// TwinCAT 3 PLC project SPS
// ProgramVersion: 3.1.4024.0
// libraries:
//   Tc2_MC2, * (Beckhoff Automation GmbH)
//   Tc2_Standard, * (Beckhoff Automation GmbH)
//   Tc2_System, * (Beckhoff Automation GmbH)
//   Tc3_IotBase, * (Beckhoff Automation GmbH)
//   Tc3_Module, * (Beckhoff Automation GmbH)
//   VisuDialogs, * (System)
//   VisuSymbols,3.5.10.0,System
// project tree:
//   DUTs/ eBetriebszustand.TcDUT (not stored)
//   / GlobalTextList.TcGTLO, PlcTask.TcTTO, Visualization Manager.TcVMO (not stored)
//   GVLs/ GVL_PosKinematic.TcGVL (not stored), IFC_HW.TcGVL (not stored)
//   POUs/Abfüllmodul/ FB_Abfuellmodul.TcPOU, FB_Dispenser.TcPOU, FB_EZylinder.TcPOU (not stored), FB_Vereinzelung.TcPOU
//   POUs/Abfüllmodul/Transport/ FB_Foerderband.TcPOU, FB_Transport.TcPOU, FB_Transport_A.TcPOU (not stored), FB_Transport_E.TcPOU (not stored), FB_Transport_Logik.TcPOU
//   POUs/ FUN_Scale.TcPOU (not stored), MAIN.TcPOU
//   POUs/IoT/ FB_MQTT.TcPOU (not stored)
//   POUs/Manipulator/ FB_Manipulator.TcPOU
//   POUs/Manipulator/Roboter/ FB_Roboter.TcPOU, FB_Roboter_Axis.TcPOU, FB_Roboter_E.TcPOU, FB_Roboter_Logik.TcPOU
//   POUs/Statusleuchte/ FB_Ampelleuchte.TcPOU (not stored), FB_Blinklicht.TcPOU (not stored)
//   VISUs/ Visualization.TcVIS
// real-time tasks:
//   TASK PlcTask: cycle T#10ms, priority 20, ADS port 350
// motion (NC):
//   TASK NC-Task 1 SAF: cycle T#2ms, priority 4, ADS port 501
//   TASK NC-Task 1 SVB: cycle T#10ms, priority 8, ADS port 511
//   AXIS Achse_Band (id 1)
//     OtherSettings: AllowMotionCmdToSlave=true
//     encoder EncType=1
//     drive DrvType=5
//       Analog: TorqueSetpointScale=10, ScaleFactorActTorque=0.1
//       TimeComp: TaskDelayCycles=1
//     controller CtrType=1
//       CtrPara: PriorControlFactor=1
//         Observer: BandWidth=20
//   AXIS Achse_Dispenser_Rot (id 2)
//     OtherSettings: AllowMotionCmdToSlave=true
//     encoder EncType=1
//     drive DrvType=5
//       Analog: TorqueSetpointScale=10, ScaleFactorActTorque=0.1
//       TimeComp: TaskDelayCycles=1
//     controller CtrType=1
//       CtrPara: PriorControlFactor=1
//         Observer: BandWidth=20
//   AXIS Achse_Dispenser_Gruen (id 3)
//     OtherSettings: AllowMotionCmdToSlave=true
//     encoder EncType=1
//     drive DrvType=5
//       Analog: TorqueSetpointScale=10, ScaleFactorActTorque=0.1
//       TimeComp: TaskDelayCycles=1
//     controller CtrType=1
//       CtrPara: PriorControlFactor=1
//         Observer: BandWidth=20
//   AXIS Achse_Dispenser_Blau (id 4)
//     OtherSettings: AllowMotionCmdToSlave=true
//     encoder EncType=1
//     drive DrvType=5
//       Analog: TorqueSetpointScale=10, ScaleFactorActTorque=0.1
//       TimeComp: TaskDelayCycles=1
//     controller CtrType=1
//       CtrPara: PriorControlFactor=1
//         Observer: BandWidth=20
//   AXIS Achse_Manipulator_X (id 5)
//     Velo: RefSearch=15, RefSync=15
//     OtherSettings: AllowMotionCmdToSlave=true
//     encoder EncType=1
//       EncPara: ScaleFactorNumerator=0.0025
//         Inc: RefSearchInverse=true, RefSyncInverse=false
//     drive DrvType=5
//       Analog: TorqueSetpointScale=10, ScaleFactorActTorque=0.1
//       TimeComp: TaskDelayCycles=1
//     controller CtrType=1
//       CtrPara: PriorControlFactor=1
//         Observer: BandWidth=20
//   AXIS Achse_Manipulator_Y (id 6)
//     Velo: RefSearch=15, RefSync=15
//     OtherSettings: AllowMotionCmdToSlave=true
//     encoder EncType=1
//       Inc: RefSearchInverse=true, RefSyncInverse=false
//     drive DrvType=5
//       Analog: TorqueSetpointScale=10, ScaleFactorActTorque=0.1
//       TimeComp: TaskDelayCycles=1
//     controller CtrType=1
//       CtrPara: PriorControlFactor=1
//         Observer: BandWidth=20
//   AXIS Achse_Manipulator_Z (id 7)
//     Velo: RefSearch=15, RefSync=15
//     OtherSettings: AllowMotionCmdToSlave=true
//     encoder EncType=1
//       Inc: RefSearchInverse=true, RefSyncInverse=false
//     drive DrvType=5
//       Analog: TorqueSetpointScale=10, ScaleFactorActTorque=0.1
//       TimeComp: TaskDelayCycles=1
//     controller CtrType=1
//       CtrPara: PriorControlFactor=1
//         Observer: BandWidth=20
//   AXIS Achse_Manipulator_Gripper (id 8)
//     OtherSettings: AllowMotionCmdToSlave=true
//     encoder EncType=1
//     drive DrvType=5
//       Analog: TorqueSetpointScale=10, ScaleFactorActTorque=0.1
//       TimeComp: TaskDelayCycles=1
//     controller CtrType=1
//       CtrPara: PriorControlFactor=1
//         Observer: BandWidth=20
// variable links:
//   SPS/SPS Instance <-> NC-Task 1 SAF/Axes/Achse_Band
//     PlcTask Inputs/IFC_HW.ax_BandMotor.NcToPlc <-> Outputs/ToPlc
//     PlcTask Outputs/IFC_HW.ax_BandMotor.PlcToNc <-> Inputs/FromPlc
//   SPS/SPS Instance <-> NC-Task 1 SAF/Axes/Achse_Dispenser_Blau
//     PlcTask Inputs/IFC_HW.ax_Extruder3.NcToPlc <-> Outputs/ToPlc
//     PlcTask Outputs/IFC_HW.ax_Extruder3.PlcToNc <-> Inputs/FromPlc
//   SPS/SPS Instance <-> NC-Task 1 SAF/Axes/Achse_Dispenser_Gruen
//     PlcTask Inputs/IFC_HW.ax_Extruder2.NcToPlc <-> Outputs/ToPlc
//     PlcTask Outputs/IFC_HW.ax_Extruder2.PlcToNc <-> Inputs/FromPlc
//   SPS/SPS Instance <-> NC-Task 1 SAF/Axes/Achse_Dispenser_Rot
//     PlcTask Inputs/IFC_HW.ax_Extruder1.NcToPlc <-> Outputs/ToPlc
//     PlcTask Outputs/IFC_HW.ax_Extruder1.PlcToNc <-> Inputs/FromPlc
//   SPS/SPS Instance <-> NC-Task 1 SAF/Axes/Achse_Manipulator_Gripper
//     PlcTask Inputs/IFC_HW.ax_ManG.NcToPlc <-> Outputs/ToPlc
//     PlcTask Outputs/IFC_HW.ax_ManG.PlcToNc <-> Inputs/FromPlc
//   SPS/SPS Instance <-> NC-Task 1 SAF/Axes/Achse_Manipulator_X
//     PlcTask Inputs/IFC_HW.ax_ManX.NcToPlc <-> Outputs/ToPlc
//     PlcTask Outputs/IFC_HW.ax_ManX.PlcToNc <-> Inputs/FromPlc
//   SPS/SPS Instance <-> NC-Task 1 SAF/Axes/Achse_Manipulator_Y
//     PlcTask Inputs/IFC_HW.ax_ManY.NcToPlc <-> Outputs/ToPlc
//     PlcTask Outputs/IFC_HW.ax_ManY.PlcToNc <-> Inputs/FromPlc
//   SPS/SPS Instance <-> NC-Task 1 SAF/Axes/Achse_Manipulator_Z
//     PlcTask Inputs/IFC_HW.ax_ManZ.NcToPlc <-> Outputs/ToPlc
//     PlcTask Outputs/IFC_HW.ax_ManZ.PlcToNc <-> Inputs/FromPlc

CONFIGURATION SPS
    RESOURCE PLC ON TwinCAT3
        TASK PlcTask(INTERVAL := T#10ms, PRIORITY := 20);
        PROGRAM MAIN WITH PlcTask : MAIN;
    END_RESOURCE
END_CONFIGURATION

// ---- POUs/MAIN.TcPOU
PROGRAM MAIN
VAR
	fb_Ampelleuchte :FB_Ampelleuchte;	
	fb_Abfuellmodul :FB_Abfuellmodul;
	fb_Manipulator :FB_Manipulator;
	
	nState :INT :=0;
	
	fb_MQTT :FB_MQTT;
END_VAR

	
fb_Ampelleuchte(eState:= , bAmpelGruen_out=> IFC_HW.bAmpelGrun, bAmpelRot_out=> IFC_HW.bAmpelRot, bAmpelGelb_out=> IFC_HW.bAmpelGelb);

fb_Abfuellmodul(bEnable:= , bExecute:= , eState=> ); 
fb_Manipulator(bEnable:= , bExecute:= , bGripperClosed=> IFC_HW.bGripperClosed, eState=> );

IF fb_Abfuellmodul.eState = eBetriebszustand.Init OR fb_Manipulator.eState = eBetriebszustand.Init THEN
	fb_Ampelleuchte.eState := eBetriebszustand.init;
ELSIF fb_Abfuellmodul.eState = eBetriebszustand.ready AND fb_Manipulator.eState = eBetriebszustand.ready THEN
	fb_Ampelleuchte.eState := eBetriebszustand.ready;
ELSIF fb_Abfuellmodul.eState = eBetriebszustand.production OR fb_Manipulator.eState = eBetriebszustand.Production THEN
	fb_Ampelleuchte.eState := eBetriebszustand.Production;
ELSIF fb_Abfuellmodul.eState = eBetriebszustand.off AND fb_Manipulator.eState = eBetriebszustand.off THEN
	fb_Ampelleuchte.eState := eBetriebszustand.off;
ELSE 
	fb_Ampelleuchte.eState := eBetriebszustand.Warning;
END_IF


IF NOT IFC_HW.bEnable THEN
	nState :=0;
END_IF
CASE nState Of
	0://off
	fb_Abfuellmodul.bEnable :=FALSE;
	fb_Manipulator.bEnable :=FALSE;
	
	IF IFC_HW.bEnable THEN
		nstate:=1;
	END_IF
	
	1: //init
	fb_Abfuellmodul.bEnable :=TRUE;
	fb_Manipulator.bEnable :=TRUE;
	
	IF fb_Abfuellmodul.eState = eBetriebszustand.Ready AND fb_Manipulator.eState = eBetriebszustand.Ready THEN
		nState:=2;
	END_IF
	
	2: //ready
	IF IFC_HW.bExecute THEN
		nstate :=21;
	END_IF
	
	21: //bottle
	fb_Abfuellmodul.bExecute :=TRUE;
	
	IF fb_Abfuellmodul.eState = eBetriebszustand.Done THEN
		fb_Abfuellmodul.bExecute :=FALSE;
		nstate :=22;
	END_IF
	
	22: //mani
	fb_Manipulator.bExecute :=TRUE;
	
	IF fb_Manipulator.eState = eBetriebszustand.Done THEN
		fb_Manipulator.bExecute :=FALSE;
		nState :=23;
	END_IF
	
	23://done
	IF NOT IFC_HW.bExecute THEN
		nState:=2;
	END_IF
END_CASE


fb_MQTT(data:= IFC_HW.bEnable);

END_PROGRAM

// ---- POUs/Abfüllmodul/FB_Abfuellmodul.TcPOU
FUNCTION_BLOCK FB_Abfuellmodul
VAR_INPUT
	bEnable :BOOL;
	bExecute :BOOL;
END_VAR
VAR_OUTPUT
	eState :eBetriebszustand;
END_VAR
VAR
	fb_Vereinzelung :FB_Vereinzelung;
	fb_Transport : FB_Transport;
	fb_Dispenser1 :FB_Dispenser;
	fb_Dispenser2 :FB_Dispenser;
	fb_Dispenser3 :FB_Dispenser;
	fb_EZylinder1 : FB_EZylinder;
	fb_EZylinder2 : FB_EZylinder;
	
	nState :INT;
	nStation :INT;
END_VAR

fb_Vereinzelung(
	bEnable:= IFC_HW.bEnable, 
	bExecute:= IFC_HW.bExecute, 
	bSens1:= IFC_HW.bEinzelSens1, 
	bSens2:= IFC_HW.bEinzelSens2, 
	bSens3:= IFC_HW.bEinzelSens3, 
	bSens4:= IFC_HW.bBandSens1, 
	eState=> , 
	bGate1=> fb_EZylinder1.bGate, 
	bGate2=> fb_EZylinder2.bGate);
	
fb_Transport(
	bEnable:= IFC_HW.bEnable, 
	bExecute:= IFC_HW.bExecute, 
	nStation:= , 
	bSens1:= IFC_HW.bBandSens1, 
	bSens2:= IFC_HW.bBandSens2, 
	bSens3:= IFC_HW.bBandSens3, 
	bSens4:= IFC_HW.bBandSens4, 
	eState=> , 
	bStopper1=> IFC_HW.bBandHub1, 
	bStopper2=> IFC_HW.bBandHub2, 
	bStopper3=> IFC_HW.bBandHub3, 
	ax:= IFC_HW.ax_BandMotor);
	
fb_Dispenser1(
	bEnable:= , 
	bExecute:= , 
	rDistance:= 60, 
	eState=> , 
	ax:= IFC_HW.ax_Extruder1);
fb_Dispenser2(
	bEnable:= , 
	bExecute:= , 
	rDistance:= 60, 
	eState=> , 
	ax:= IFC_HW.ax_Extruder2);
fb_Dispenser3(
	bEnable:= , 
	bExecute:= , 
	rDistance:= 60, 
	eState=> , 
	ax:= IFC_HW.ax_Extruder3);


CASE nState OF
	0: // Off
	eState := eBetriebszustand.Off;
	
	fb_Vereinzelung.bEnable:=FALSE;
	fb_Transport.bEnable :=FALSE;
	fb_Dispenser1.bEnable :=FALSE;
	fb_Dispenser2.bEnable :=FALSE;
	fb_Dispenser3.bEnable :=FALSE;
	fb_Vereinzelung.bExecute :=FALSE;
	fb_Transport.bExecute :=FALSE;
	fb_Dispenser1.bExecute :=FALSE;
	fb_Dispenser2.bExecute :=FALSE;
	fb_Dispenser3.bExecute :=FALSE;
	
	IF bEnable THEN
		nstate :=10;
	END_IF
	
	10:// Init
	eState := eBetriebszustand.Init;
	
	fb_Vereinzelung.bEnable:=TRUE;
	fb_Transport.bEnable :=TRUE;
	fb_Dispenser1.bEnable :=TRUE;
	fb_Dispenser2.bEnable :=TRUE;
	fb_Dispenser3.bEnable :=TRUE;
	fb_Vereinzelung.bExecute :=FALSE;
	fb_Transport.bExecute :=FALSE;
	fb_Dispenser1.bExecute :=FALSE;
	fb_Dispenser2.bExecute :=FALSE;
	fb_Dispenser3.bExecute :=FALSE;
	
	IF (fb_Vereinzelung.eState = eBetriebszustand.Ready) AND (fb_Transport.eState = eBetriebszustand.Ready) AND (fb_Dispenser1.eState = eBetriebszustand.Ready) AND (fb_Dispenser2.eState = eBetriebszustand.Ready) AND (fb_Dispenser3.eState = eBetriebszustand.Ready)THEN
		nstate :=20;
	END_IF
	
	20:// Ready
	eState := eBetriebszustand.Ready;
	
	fb_Vereinzelung.bEnable:=TRUE;
	fb_Transport.bEnable :=TRUE;
	fb_Dispenser1.bEnable :=TRUE;
	fb_Dispenser2.bEnable :=TRUE;
	fb_Dispenser3.bEnable :=TRUE;
	fb_Vereinzelung.bExecute :=FALSE;
	fb_Transport.bExecute :=FALSE;
	fb_Dispenser1.bExecute :=FALSE;
	fb_Dispenser2.bExecute :=FALSE;
	fb_Dispenser3.bExecute :=FALSE;
	
	IF bExecute THEN
		nState:=30;
	END_IF
	
	30:// Start
	eState := eBetriebszustand.Production;
	
	//fb_Vereinzelung.bEnable:=TRUE;
	//fb_Transport.bEnable :=TRUE;
	//fb_Dispenser1.bEnable :=TRUE;
	//fb_Dispenser2.bEnable :=TRUE;
	//fb_Dispenser3.bEnable :=TRUE;
	fb_Vereinzelung.bExecute :=TRUE;
	fb_Transport.bExecute :=TRUE;
	fb_Dispenser1.bExecute :=FALSE;
	fb_Dispenser2.bExecute :=FALSE;
	fb_Dispenser3.bExecute :=FALSE;
	nstation :=1;
	
	IF (fb_Vereinzelung.eState = eBetriebszustand.Done) AND (fb_Transport.eState = eBetriebszustand.Done) THEN
		nstate :=31;
	END_IF
	
	31:// Dispenser1
	eState := eBetriebszustand.Production;
	
	//fb_Vereinzelung.bEnable:=TRUE;
	//fb_Transport.bEnable :=TRUE;
	//fb_Dispenser1.bEnable :=TRUE;
	//fb_Dispenser2.bEnable :=TRUE;
	//fb_Dispenser3.bEnable :=TRUE;
	fb_Vereinzelung.bExecute :=FALSE;
	fb_Transport.bExecute :=FALSE;
	fb_Dispenser1.bExecute :=TRUE;
	fb_Dispenser2.bExecute :=FALSE;
	fb_Dispenser3.bExecute :=FALSE;
	nstation :=1;
	
	IF fb_Dispenser1.eState = eBetriebszustand.Done THEN
		nState :=32;
	END_IF
	
	32:// Bewegung zu Dispenser2
	eState := eBetriebszustand.Production;
	
	nstation :=2;
	fb_Vereinzelung.bExecute :=FALSE;
	fb_Transport.bExecute :=TRUE;
	fb_Dispenser1.bExecute :=FALSE;
	fb_Dispenser2.bExecute :=FALSE;
	fb_Dispenser3.bExecute :=FALSE;
	
	IF fb_Transport.eState = eBetriebszustand.Done THEN
		nState :=33;
	END_IF
	
	33:// Dispenser2
	eState := eBetriebszustand.Production;
	
	fb_Vereinzelung.bExecute :=FALSE;
	fb_Transport.bExecute :=FALSE;
	fb_Dispenser1.bExecute :=FALSE;
	fb_Dispenser2.bExecute :=TRUE;
	fb_Dispenser3.bExecute :=FALSE;
	nstation :=2;
	
	IF fb_Dispenser2.eState = eBetriebszustand.Done THEN
		nState :=34;
	END_IF
		
	34:// Bewegung zu Dispenser3
	eState := eBetriebszustand.Production;
	
	nstation :=3;
	fb_Vereinzelung.bExecute :=FALSE;
	fb_Transport.bExecute :=TRUE;
	fb_Dispenser1.bExecute :=FALSE;
	fb_Dispenser2.bExecute :=FALSE;
	fb_Dispenser3.bExecute :=FALSE;
	
	IF fb_Transport.eState = eBetriebszustand.Done THEN
		nState :=35;
	END_IF
	
	35:// Dispenser3
	eState := eBetriebszustand.Production;
	
	fb_Vereinzelung.bExecute :=FALSE;
	fb_Transport.bExecute :=FALSE;
	fb_Dispenser1.bExecute :=FALSE;
	fb_Dispenser2.bExecute :=FALSE;
	fb_Dispenser3.bExecute :=TRUE;
	nstation :=3;
	
	IF fb_Dispenser3.eState = eBetriebszustand.Done THEN
		nState :=36;
	END_IF
	
	36:// Abholstation
	eState := eBetriebszustand.Production;
	
	nstation :=4;
	fb_Vereinzelung.bExecute :=FALSE;
	fb_Transport.bExecute :=TRUE;
	fb_Dispenser1.bExecute :=FALSE;
	fb_Dispenser2.bExecute :=FALSE;
	fb_Dispenser3.bExecute :=FALSE;
		
	IF fb_Transport.eState = eBetriebszustand.Done THEN
		nState :=40;
	END_IF 
	
	40:// Done
	eState := eBetriebszustand.Done;
	
	fb_Vereinzelung.bExecute :=FALSE;
	fb_Transport.bExecute :=FALSE;
	fb_Dispenser1.bExecute :=FALSE;
	fb_Dispenser2.bExecute :=FALSE;
	fb_Dispenser3.bExecute :=FALSE;
	
	IF NOT bExecute THEN
		nState :=30;
	END_IF
	
	
END_CASE

END_FUNCTION_BLOCK

// ---- POUs/Abfüllmodul/FB_Vereinzelung.TcPOU
FUNCTION_BLOCK FB_Vereinzelung
VAR_INPUT
	//Steuervariablen
	bEnable :BOOL;
	bExecute :BOOL;
	
	//Hardwareeingänge
	bSens1 :BOOL; //Flasche in der Kammer
	bSens2 :BOOL; //Flasche im Rohr
	bSens3 :BOOL; //Flasche verkehrt
	bSens4 :BOOL; //Flasche am Förderband
END_VAR
VAR_OUTPUT
	//Steuervariable 
	eState :eBetriebszustand;
	
	//Hardwareausgägne
	bGate1 :BOOL;
	bGate2 :BOOL;
END_VAR
VAR
	nState :INT :=100;
	fbTON :TON;
END_VAR

fbTON(IN:= , PT:= T#2S, Q=> , ET=> );

IF NOT bEnable THEN
	nState :=0;
END_IF

CASE nState OF
	100: //Off oder nicht BEtriebsbereit 
	eState:=eBetriebszustand.Off;
	
	IF bSens1 AND bEnable THEN
		nState:=21; //Ready
	ELSIF bEnable THEN
		nState :=0; //Init
	END_IF
	
	
	0: //Kammer ist leer
	eState:=eBetriebszustand.Init;
	
	bGate1:=FALSE;
	bGate2:=FALSE;
	
	IF bSens2 THEN
		nState:=1; //Oben öffnen
	END_IF
	
	
	1: //Oben öffnen
	eState := eBetriebszustand.Init;
	
	bGate1:=TRUE;
	bGate2 :=FALSE;
	
	IF bSens1 THEN
		nState:=2; //Oben schleißen
	END_IF
	
	
	2: //Oben schließen
	eState := eBetriebszustand.Init;
	
	bGate1:=FALSE;
	bGate2 :=FALSE;
	fbTon.IN:=TRUE;
	
	IF fbTon.Q THEN
		nState:=21; //Ready
		fbTon.IN :=FALSE;
	END_IF
	
	21: //Ready
	eState := eBetriebszustand.Ready;
	
	bGate1:=FALSE;
	bGate2 :=FALSE;
	
	IF bExecute THEN
		nState:=3; //Unten öffnen
	END_IF
	
	
	3: //Unten öffnen
	eState := eBetriebszustand.Production;
	
	bGate1:=FALSE;
	bGate2 :=TRUE;
	
	IF bSens4 THEN
		nState :=4; //Unten schließen
	END_IF
	
	4: //Unten schließen
	eState := eBetriebszustand.Production;
	
	bGate1:=FALSE;
	bGate2 :=FALSE;
	fbTon.IN :=TRUE;
	
	IF fbTon.Q THEN
		nState:=41; //Done
		fbTon.IN :=FALSE;
	END_IF
	
	41: //Done
	eState:= eBetriebszustand.Done;
	
	IF NOT bExecute THEN
		nState :=0; //Kammer leer
	END_IF
	
	
END_CASE

END_FUNCTION_BLOCK

// ---- POUs/Abfüllmodul/Transport/FB_Transport.TcPOU
FUNCTION_BLOCK FB_Transport
VAR_INPUT
	bEnable :BOOL;
	bExecute :BOOL;
	nStation :INT := 1;
	//Hardweare Eingänge
	bSens1 :BOOL;
	bSens2 :BOOL;
	bSens3 :BOOL;
	bSens4 :BOOL;
END_VAR
VAR_OUTPUT
	eState :eBetriebszustand;
	bStopper1 :BOOL;
	bStopper2 :BOOL;
	bStopper3 :BOOL;
END_VAR
VAR
	fb_TransportE :FB_Transport_E;
	fb_TransportLogik :FB_Transport_Logik;
	fb_TransportBand :FB_Foerderband;
	fb_TransportA :FB_Transport_A;
END_VAR
VAR_IN_OUT
	//Achsen Ref
	ax : AXIS_REF;
END_VAR

//nur Eingänge werden beschreiben 
fb_TransportE(
	bSens1:= bSens1, 
	bSens2:= bSens2, 
	bSens3:= bSens3, 
	bSens4:= bSens4, 
	bStation1=> , 
	bStation2=> , 
	bStation3=> , 
	bStation4=> );
	
fb_TransportLogik(
	bEnable:= bEnable, 
	bExecute:= bExecute, 
	eStateE:= fb_TransportBand.eState, 
	nStation:= nStation, 
	bStation1:= fb_TransportE.bStation1, 
	bStation2:= fb_TransportE.bStation2, 
	bStation3:= fb_TransportE.bStation3, 
	bStation4:= fb_TransportE.bStation4,
	bEnableA=> , 
	bExecuteA=> , 
	bStopA=> , 
	eStateA=> eState, 
	bStop1=> , 
	bStop2=> , 
	bStop3=> );
	
	
fb_TransportBand(
	bEnable:= fb_TransportLogik.bEnableA, 
	bExecute:= fb_TransportLogik.bExecuteA, 
	bHalt:= fb_TransportLogik.bStopA, 
	eState=> , 
	ax:= ax);
	
	
fb_TransportA(
	bStop1:= fb_TransportLogik.bStop1, 
	bStop2:= fb_TransportLogik.bStop2, 
	bStop3:= fb_TransportLogik.bStop3, 
	bStopper1=> bStopper1, 
	bStopper2=> bStopper2, 
	bStopper3=> bStopper3);

END_FUNCTION_BLOCK

// ---- POUs/Abfüllmodul/Transport/FB_Transport_Logik.TcPOU
FUNCTION_BLOCK FB_Transport_Logik
VAR_INPUT
	bEnable :BOOL;
	bExecute :BOOL;
	eStateE :eBetriebszustand;
	nStation :INT;
	//Logik -> Hardware Signale
	bStation1 :BOOL;
	bStation2 :BOOL;
	bStation3 :BOOL;
	bStation4 :BOOL;
END_VAR
VAR_OUTPUT
	bEnableA :BOOL;
	bExecuteA :BOOL;
	bStopA :BOOL;
	eStateA :eBetriebszustand;
	
	//Hardware Singale ->Logik
	bStop1 :BOOL;
	bStop2 :BOOL;
	bStop3 :BOOL;
END_VAR
VAR
	nState :INT;
	
END_VAR

//Zustandsgraphen aus PP selber gezeichent implementieren 

IF NOT bEnable THEN
	nState :=0;
END_IF

CASE nState OF 
	0: //off
	eStateA:= eBetriebszustand.Off;
	bEnableA :=FALSE;
	bExecuteA :=FALSE;
	bStopA :=FALSE;
	bStop1 :=FALSE;
	bStop2 :=FALSE;
	bStop3 :=FALSE;
	
	IF bEnable THEN 
		nState :=1;
	END_IF

	1: //init
	eStateA:=eBetriebszustand.Init;
	bEnableA :=TRUE;
	bExecuteA :=FALSE;
	bStopA :=FALSE;
	bStop1 :=FALSE;
	bStop2 :=FALSE;
	bStop3 :=FALSE;
	
	IF eStateE = eBetriebszustand.Ready THEN
		nState :=2;
	END_IF
	
	2: //Ready
	eStateA:=eBetriebszustand.Ready;
	bEnableA :=TRUE;
	bExecuteA :=FALSE;
	bStopA :=FALSE;
	bStop1 :=FALSE;
	bStop2 :=FALSE;
	bStop3 :=FALSE;
	
	IF bExecute THEN
		nState :=3;
	END_IF
	
	3: //Förderband Start
	eStateA:=eBetriebszustand.Production;
	bExecuteA :=TRUE;
	
	IF (nStation-1) = 1 THEN
		bStop1 :=TRUE;
	ELSIF (nStation-1) = 2 THEN
		bStop2 :=TRUE;		
	ELSIF (nStation-1) = 3 THEN
		bStop3 :=TRUE;		
	END_IF
	
	IF (bStation1 AND (nStation =1)) OR (bStation2 AND (nStation =2)) OR (bStation3 AND (nStation =3)) OR (bStation4 AND (nStation =4))THEN
		nState :=4;
	END_IF
	
	4: //Förderband stop
	eStateA:=eBetriebszustand.Production;
	bExecuteA := FALSE;
	bStopA := TRUE;
	bStop1 :=FALSE;
	bStop2 :=FALSE;
	bStop3 :=FALSE;
	
	IF eStateE = eBetriebszustand.Done THEN
		nState :=5;
	END_IF
	
	5: //Done
	eStateA:=eBetriebszustand.Done;
	
	IF NOT bExecute THEN
		nState :=2;
	END_IF
END_CASE

END_FUNCTION_BLOCK

// ---- POUs/Abfüllmodul/Transport/FB_Foerderband.TcPOU
FUNCTION_BLOCK FB_Foerderband
VAR_INPUT
	bEnable :BOOL;
	bExecute :BOOL;
	bHalt :BOOL;
END_VAR
VAR_OUTPUT
	eState :eBetriebszustand;
END_VAR
VAR
	nState:INT :=0;
	mc_Reset :MC_Reset;
	mc_Velocity :MC_MoveVelocity;
	mc_Halt :MC_Halt;
	mc_Power :MC_Power;
	Timer :TON;
END_VAR
VAR_IN_OUT
	ax : Axis_Ref;
END_VAR

ax.ReadStatus();
mc_Reset(
	Axis:= ax, 
	Execute:= , 
	Done=> , 
	Busy=> , 
	Error=> , 
	ErrorID=> );
	
mc_Power(
	Axis:= ax, 
	Enable:= , 
	Enable_Positive:= , 
	Enable_Negative:= , 
	Override:= , 
	BufferMode:= , 
	Options:= , 
	Status=> , 
	Busy=> , 
	Error=> , 
	ErrorID=> );
	
mc_Velocity(
	Axis:= ax, 
	Execute:= , 
	Velocity:= 30, 
	Acceleration:= 60, 
	Deceleration:= 60, 
	Jerk:= , 
	Direction:= MC_Positive_Direction, 
	BufferMode:= , 
	Options:= , 
	InVelocity=> , 
	Busy=> , 
	Active=> , 
	CommandAborted=> , 
	Error=> , 
	ErrorID=> );
	
mc_Halt(
	Axis:= ax, 
	Execute:= , 
	Deceleration:= 60, 
	Jerk:= , 
	BufferMode:= , 
	Options:= , 
	Done=> , 
	Busy=> , 
	Active=> , 
	CommandAborted=> , 
	Error=> , 
	ErrorID=> );
	
Timer(IN:= , PT:= T#1S, Q=> , ET=> );


//Originalcode funktioniert wenn hier die Flanke kontrolliert wird 
//Anstelle vom Power.Status
//IF NOT mc_Power.Status THEN
//	nState:=0;
//END_IF

IF NOT bEnable THEN
	nState :=0;
END_IF

CASE nState OF 
	0:
	eState:=eBetriebszustand.Off;
	mc_power.Enable :=TRUE;
	mc_Power.Enable_Positive :=TRUE;
	
	IF bEnable AND NOT mc_power.Status THEN
		nState :=10;
	ELSIF mc_power.Status AND bEnable THEN
		nState:=20;
	END_IF
	
	10: // init Reset
	eState:=eBetriebszustand.Init;
	
	//nicht power resetten sonst durch if vor case in dauerschleife zwischen 0 und 11
	//mc_Power.Enable:=FALSE;
	//mc_Power.Enable_Positive:=FALSE;
	
	mc_Reset.Execute:=TRUE;
	
	IF mc_Reset.Done THEN
		nState:=11;
		mc_Reset.Execute:=FALSE;
	END_IF
	
	11: // init Power
	eState:=eBetriebszustand.Init;
	mc_Power.Enable:=TRUE;
	mc_Power.Enable_Positive :=TRUE;
	
	IF mc_Power.Status THEN
		nState:=20;
	END_IF
	
	20: // Ready
	eState:= eBetriebszustand.Ready;
	
	IF bExecute THEN 
		nState:=30;
	END_IF
 
	30: // Kontinuierliche Bewegung
	eState:=eBetriebszustand.Production;
	mc_Velocity.Execute:=TRUE;
	
	IF bHalt THEN 
		nState :=31;
	END_IF
	
	31: //TON verzögerung dass flasche noch bis zum anschlag fährt
	eState :=eBetriebszustand.Production;
	Timer.IN:=TRUE;
	
	IF Timer.Q THEN
		nState:=32;
		Timer.IN:=FALSE;
	END_IF
	
	32: //Halten
	eState := eBetriebszustand.Production;
	mc_Velocity.Execute:=FALSE;
	mc_Halt.Execute:=TRUE;
	
	IF mc_Halt.Done THEN 
		nState:=40;
	END_IF
	
	40: // Fertig
	eState :=eBetriebszustand.Done;
	mc_halt.Execute:=FALSE;
	
	IF NOT bExecute THEN 
		nState:=20;
	END_IF
END_CASE

END_FUNCTION_BLOCK

// ---- POUs/Abfüllmodul/FB_Dispenser.TcPOU
FUNCTION_BLOCK FB_Dispenser
VAR_INPUT
	bEnable :BOOL;
	bExecute :BOOL;
	rDistance :REAL;
END_VAR
VAR_OUTPUT
	eState :eBetriebszustand;
END_VAR
VAR
	mc_Reset :MC_Reset;
	mc_Power :MC_Power;
	mc_MoveRelative :MC_MoveRelative;
	nState :INT :=0;
END_VAR
VAR_IN_OUT
	ax :Axis_Ref;
END_VAR

ax.ReadStatus();
mc_Reset(
	Axis:= ax, 
	Execute:= , 
	Done=> , 
	Busy=> , 
	Error=> , 
	ErrorID=> );
	
mc_Power(
	Axis:= ax, 
	Enable:= , 
	Enable_Positive:= , 
	Enable_Negative:= , 
	Override:= , 
	BufferMode:= , 
	Options:= , 
	Status=> , 
	Busy=> , 
	Error=> , 
	ErrorID=> );
	
mc_MoveRelative(
	Axis:= ax, 
	Execute:= , 
	Distance:= rDistance, 
	Velocity:= 60, 
	Acceleration:= 30, 
	Deceleration:= 30, 
	Jerk:= , 
	BufferMode:= , 
	Options:= , 
	Done=> , 
	Busy=> , 
	Active=> , 
	CommandAborted=> , 
	Error=> , 
	ErrorID=> );
	

//IF NOT mc_Power.Status THEN
//	nState:=0;
//END_IF

IF NOT bEnable THEN
	nState:=0;
END_IF

CASE nState OF 
	0:
	eState:=eBetriebszustand.Off;
	mc_Power.Enable :=TRUE;
	mc_Power.Enable_Positive:=TRUE;
	
	
	IF bEnable AND NOT mc_power.Status THEN
		nState :=10;
	ELSIF mc_power.Status AND bEnable THEN
		nState:=20;
	END_IF
	
	10: // init Reset
	eState:=eBetriebszustand.Init;
	mc_Reset.Execute:=TRUE;
	//mc_Power.Enable:=FALSE;
	
	IF mc_Reset.Done THEN
		nState:=11;
	END_IF
	
	11: // init Power
	eState:=eBetriebszustand.Init;
	mc_Reset.Execute:=FALSE;
	mc_Power.Enable :=TRUE;
	mc_Power.Enable_Positive:=TRUE;
	
	
	IF mc_Power.Status THEN
		nState:=20;
	END_IF
	
	20: // Ready
	eState:= eBetriebszustand.Ready;
	
	IF bExecute THEN 
		nState:=30;
	END_IF
 
	30: // Kontinuierliche Bewegung
	eState:=eBetriebszustand.Production;
	mc_MoveRelative.Execute :=TRUE;
	
	IF mc_MoveRelative.Done THEN 
		mc_MoveRelative.Execute:=FALSE;
		nState :=40;
	END_IF
	
	40: // Fertig
	eState :=eBetriebszustand.Done;
	
	IF NOT bExecute THEN 
		nState:=20;
	END_IF

END_CASE

END_FUNCTION_BLOCK

// ---- POUs/Manipulator/FB_Manipulator.TcPOU
FUNCTION_BLOCK FB_Manipulator
VAR_INPUT
	bEnable :BOOL; 
	bExecute :BOOL; //Sensor band 
END_VAR
VAR_OUTPUT
	bGripperClosed :BOOL;
	eState :eBetriebszustand;
END_VAR
VAR
	fb_Roboter :FB_Roboter;
	fb_Roboter_Gripper : FB_Roboter_Axis;
	fb_Gripper_E :FB_Roboter_E;
	//FB_waage
	//FB temp
	
	
	nState :INT :=0;
	nStation :INT :=0; 
	pPositionX :REAL;
	pPositionY :REAL;
	pPositionZ :REAL;
	
	
	
	
	nBottles: INT :=0;
END_VAR

fb_Roboter(
	bEnable:= , 
	bExecute:= , 
	pPositionX:= pPositionX, 
	pPositionY:= pPositionY, 
	pPositionZ:= pPositionZ, 
	eState=> );
	
fb_Gripper_E(bRefMax_in:= bManEndGmax, bRefMin_in:= bManEndGmin, bRefMax_out=> , bRefMin_out=> );
fb_Roboter_Gripper(
	bEnable:= , 
	bExecute:= , 
	rPosition:= , 
	bRefSens:= fb_Gripper_E.bRefMin_out, 
	eState=> , 
	ax:= IFC_HW.ax_ManG);
	
IF NOT bEnable THEN
	nState :=0;
END_IF	
	
	
CASE nState OF 
	0: //off
	eState:=eBetriebszustand.Off;
	IF bEnable THEN
		nState:=1;
	END_IF
	
	1: //init
	eState:=eBetriebszustand.Init;
	nbottles :=0;
	fb_Roboter_Gripper.bEnable:=TRUE;
	fb_Roboter.bEnable :=TRUE;
	
	IF (fb_Roboter_Gripper.eState = eBetriebszustand.Ready) AND (fb_Roboter.eState = eBetriebszustand.Ready) THEN 
		nState:=2;
	END_IF
	
	2://home //vlt auch heir 2
	eState:=eBetriebszustand.Init;
	nStation :=0;
	fb_Roboter.bExecute :=TRUE;
	fb_Roboter_Gripper.rPosition := 7; //offen;
	fb_Roboter_Gripper.bExecute :=TRUE;
	bGripperClosed :=FALSE;
	
	IF (fb_Roboter_Gripper.eState = eBetriebszustand.Done) AND (fb_Roboter.eState = eBetriebszustand.Done) THEN 
		fb_Roboter.bExecute :=FALSE;
		fb_Roboter_Gripper.bExecute :=FALSE;
		nState:=20;
	END_IF
	
	20: //Ready
	IF nstation =7 THEN
		eState:=eBetriebszustand.Stop;
		//zusätzlicher state  bei dem man nur mit quittierung rauskommt 
	ELSE
			eState:=eBetriebszustand.Ready;
	END_IF
	
	nStation :=0;
	
	IF bExecute THEN 
		nState:=21;
	END_IF
	
	21: //open gripper
	eState:=eBetriebszustand.Production;
	fb_Roboter_Gripper.rPosition := 7; //offen;
	fb_Roboter_Gripper.bExecute :=TRUE;
	bGripperClosed :=FALSE;
	
	IF fb_Roboter_Gripper.eState = eBetriebszustand.Done THEN 
		fb_Roboter_Gripper.bExecute :=FALSE;
		nState:=22;
		
	END_IF
	
	22: //move to position
	eState:= eBetriebszustand.Production;
	nstation := 1;
	fb_Roboter.bExecute :=TRUE;
	
	IF fb_Roboter.eState = eBetriebszustand.Done THEN
		fb_Roboter.bExecute :=FALSE;
		nstate:=23;
	END_IF
	
	23: //close Gripper
	eState:=eBetriebszustand.Production;
	fb_Roboter_Gripper.rPosition := 19.4; //geschlossen;
	fb_Roboter_Gripper.bExecute :=TRUE;
	bGripperClosed :=TRUE;
	
	IF fb_Roboter_Gripper.eState = eBetriebszustand.Done THEN 
		fb_Roboter_Gripper.bExecute :=FALSE;
		nState:=24;
		nstation := nStation+1;
	END_IF
	
	24://move to new position
	eState:= eBetriebszustand.Production;
	
	fb_Roboter.bExecute :=TRUE;
	
	IF fb_Roboter.eState = eBetriebszustand.Done THEN
		fb_Roboter.bExecute :=FALSE;
		nstate:=25;
	END_IF
	
	25: //open gripper
	eState:=eBetriebszustand.Production;
	fb_Roboter_Gripper.rPosition := 7; //offen;
	fb_Roboter_Gripper.bExecute :=TRUE;
	bGripperClosed :=FALSE;
	
	IF fb_Roboter_Gripper.eState = eBetriebszustand.Done THEN 
		fb_Roboter_Gripper.bExecute :=FALSE;
		nState:=26;
	END_IF
	
	26: //do Position
	eState:=eBetriebszustand.Production;
	IF nStation >3 THEN
		nbottles := nBottles +1;
		nstate :=27;
	ELSIF nStation =3 THEN
		//wait
		nStation:= nstation +nBottles;
		nstate :=23;
	ELSIF nstation =2 THEN
		//wait
		nstate :=23;
	ELSE 
		nstate :=23;
	END_IF
	
	27: //Done
	eState:=eBetriebszustand.Done;
	IF NOT bExecute THEN 
		nstate:=2;
	END_IF
END_CASE



CASE nStation OF
	0: //Home
	pPositionX :=GVL_PosKinematic.pXhome;
	pPositionY :=GVL_PosKinematic.pYhome;
	pPositionZ :=GVL_PosKinematic.pZhome;
	//fb home
	
	1: //Conveyor
	pPositionX :=GVL_PosKinematic.pXconv;
	pPositionY :=GVL_PosKinematic.pYconv;
	pPositionZ:=GVL_PosKinematic.pZconv;
	//Fbconvoyer
	
	2: //Scale
	pPositionX :=GVL_PosKinematic.pXscale;
	pPositionY :=GVL_PosKinematic.pYscale;
	pPositionZ:=GVL_PosKinematic.pZscale;
	//scale wait
	
	3: //Heating
	pPositionX :=GVL_PosKinematic.pXheat;
	pPositionY :=GVL_PosKinematic.pYheat;
	pPositionZ:=GVL_PosKinematic.pZheat;
	//fb heating
	
	4: //storage1
	pPositionX :=GVL_PosKinematic.pX1stor;
	pPositionY :=GVL_PosKinematic.pYstor;
	pPositionZ:=GVL_PosKinematic.pZstor;
	
	5: //storage2
	pPositionX :=GVL_PosKinematic.pX2stor;
	pPositionY :=GVL_PosKinematic.pYstor;
	pPositionZ:=GVL_PosKinematic.pZstor;
	
	6: //storage3
	pPositionX :=GVL_PosKinematic.pX3stor;
	pPositionY :=GVL_PosKinematic.pYstor;
	pPositionZ:=GVL_PosKinematic.pZstor;
	
	7: //storage4
	pPositionX :=GVL_PosKinematic.pX4stor;
	pPositionY :=GVL_PosKinematic.pYstor;
	pPositionZ:=GVL_PosKinematic.pZstor;
	
	
END_CASE

END_FUNCTION_BLOCK

// ---- POUs/Manipulator/Roboter/FB_Roboter.TcPOU
FUNCTION_BLOCK FB_Roboter
VAR_INPUT
END_VAR
VAR_OUTPUT
END_VAR
VAR
END_VAR

END_FUNCTION_BLOCK

// ---- POUs/Manipulator/Roboter/FB_Roboter_Axis.TcPOU
FUNCTION_BLOCK FB_Roboter_Axis
VAR_INPUT
	bEnable :BOOL;
	bExecute :BOOL;
	rPosition :REAL;
	bRefSens :BOOL;
END_VAR
VAR_OUTPUT
	eState :eBetriebszustand;
END_VAR
VAR
	nState:INT :=0;
	mc_Reset :MC_Reset;
	mc_MoveAbsolute :MC_MoveAbsolute;
	mc_Home :MC_Home;
	mc_Power :MC_Power;
	mc_HomingMode1: MC_HomingMode;
	
END_VAR
VAR_IN_OUT
	ax :AXIS_REF;
END_VAR

ax.ReadStatus();


mc_Home(
	Axis:= ax, 
	Execute:= , 
	Position:= 0, 
	HomingMode:= mc_HomingMode1, 
	BufferMode:= , 
	Options:= , 
	bCalibrationCam:= bRefSens, 
	Done=> , 
	Busy=> , 
	Active=> , 
	CommandAborted=> , 
	Error=> , 
	ErrorID=> );
	
mc_MoveAbsolute(
	Axis:= ax, 
	Execute:= , 
	Position:= , 
	Velocity:= 30, 
	Acceleration:= 30, 
	Deceleration:= 30, 
	Jerk:= , 
	BufferMode:= , 
	Options:= , 
	Done=> , 
	Busy=> , 
	Active=> , 
	CommandAborted=> , 
	Error=> , 
	ErrorID=> );

mc_Power(
	Axis:= ax, 
	Enable:= , 
	Enable_Positive:= , 
	Enable_Negative:= , 
	Override:= , 
	BufferMode:= , 
	Options:= , 
	Status=> , 
	Busy=> , 
	Error=> , 
	ErrorID=> );
	
mc_Reset(
	Axis:= ax, 
	Execute:= , 
	Done=> , 
	Busy=> , 
	Error=> , 
	ErrorID=> );
	
//IF NOT mc_Power.Status THEN
//	nState:=0;
//END_IF

IF NOT bEnable THEN
	nState :=0;
END_IF

CASE nState OF 
	0:
	eState:=eBetriebszustand.Off;
	mc_Power.Enable :=TRUE;
	mc_Power.Enable_Positive := TRUE;  
	mc_Power.Enable_Negative := TRUE;

	
	
	IF bEnable AND NOT mc_power.Status THEN
		nState :=10;
	ELSIF mc_power.Status AND bEnable THEN
		nState:=12;
	END_IF
	
	10: // init Reset
	eState:=eBetriebszustand.Init;
	mc_Reset.Execute:=TRUE;
	//mc_Power.Enable:=FALSE;
	
	IF mc_Reset.Done THEN
		nState:=11;
		mc_Reset.Execute:=FALSE;
	END_IF
	
	11: // init Power
	eState:=eBetriebszustand.Init;
	
	mc_Power.Enable :=TRUE;
	//mc_Power.Enable_Positive:=TRUE;
	
	
	IF mc_Power.Status THEN
		nState:=12;
	END_IF
	
	12://Homed?
	eState:=eBetriebszustand.Init;
	
	IF ax.Status.Homed THEN
		nstate:=20;
	ELSE
		nstate:=13;
	END_IF
	
	13://Homing
	eState:=eBetriebszustand.Init;
	
	mc_Home.Execute :=TRUE;
	
	IF mc_Home.Done THEN
		mc_Home.Execute :=FALSE;
		nstate:= 20;
	END_IF
	
	
	20: // Ready
	eState:= eBetriebszustand.Ready;
	
	IF bExecute THEN 
		nState:=30;
	END_IF
 
	30: // Bewegung
	eState:=eBetriebszustand.Production;
	mc_MoveAbsolute.Position := rPosition;
	mc_MoveAbsolute.Execute :=TRUE;
	
	IF mc_MoveAbsolute.Done THEN 
		mc_MoveAbsolute.Execute:=FALSE;
		nState :=40;
	END_IF
	
	40: // Fertig
	eState :=eBetriebszustand.Done;
	
	IF NOT bExecute THEN 
		nState:=20;
	END_IF

END_CASE

END_FUNCTION_BLOCK

// ---- POUs/Manipulator/Roboter/FB_Roboter_E.TcPOU
FUNCTION_BLOCK FB_Roboter_E
VAR_INPUT
END_VAR
VAR_OUTPUT
END_VAR
VAR
END_VAR

END_FUNCTION_BLOCK

// ---- POUs/Manipulator/Roboter/FB_Roboter_Logik.TcPOU
FUNCTION_BLOCK FB_Roboter_Logik
VAR_INPUT
	bEnable :BOOL;
	bExecute :BOOL;

	pPositionX :REAL;
	bRefmin_X :BOOL;
	bRefmax_X :BOOL;
	
	pPositionY :REAL;
	bRefmin_Y :BOOL;
	bRefmax_Y :BOOL;
	
	pPositionZ :REAL;
	bRefmin_Z :BOOL;
	bRefmax_Z :BOOL;
	
	
	
	
END_VAR
VAR_OUTPUT
	bBreak :BOOL;
	
	
	eState :eBetriebszustand;
	
END_VAR
VAR
	fb_Roboter_Axis_X : FB_Roboter_Axis;
	fb_Roboter_Axis_Y : FB_Roboter_Axis;
	fb_Roboter_Axis_Z : FB_Roboter_Axis;
	//fb_Roboter_Gripper : FB_Roboter_Axis;
	
	nState :INT;
END_VAR

//endschlter prüfen in axis noch hinzufügen 
//soft limits bei achse einstellen 

fb_Roboter_Axis_X(
	bEnable:= , 
	bExecute:= , 
	rPosition:= , 
	bRefSens:= bRefmin_X, 
	eState=> , 
	ax:= IFC_HW.ax_ManX);
fb_Roboter_Axis_Y(
	bEnable:= , 
	bExecute:= , 
	rPosition:= , 
	bRefSens:= bRefmin_Y, 
	eState=> , 
	ax:= IFC_HW.ax_ManY);
fb_Roboter_Axis_Z(
	bEnable:= , 
	bExecute:= , 
	rPosition:= , 
	bRefSens:= bRefmin_Z, 
	eState=> , 
	ax:= IFC_HW.ax_ManZ);

IF NOT bEnable THEN
	nState :=0;
END_IF

CASE nState OF
	0: //off
	eState := eBetriebszustand.Off;
	
	IF bEnable THEN
		nstate :=1;
	END_IF
	
	1: //init
	eState := eBetriebszustand.Init;
	fb_Roboter_Axis_X.bEnable := TRUE;
	fb_Roboter_Axis_Y.bEnable := TRUE;
	fb_Roboter_Axis_Z.bEnable := TRUE;
	
	IF (fb_Roboter_Axis_X.eState = eBetriebszustand.Ready) AND (fb_Roboter_Axis_Y.eState = eBetriebszustand.Ready) AND (fb_Roboter_Axis_Z.eState = eBetriebszustand.Ready) THEN 
		nstate :=2;
	END_IF
	
	2: //Ready
	eState := eBetriebszustand.Ready;
	
	IF bExecute THEN 
		nstate :=21;
	END_IF
	
	21: //check z hight
	eState := eBetriebszustand.Production;
	
	IF IFC_HW.ax_ManZ.NcToPlc.ActPos > GVL_PosKinematic.pZoff THEN
		nstate :=22;
	ELSE
		nstate :=23;
	END_IF
	
	22: //Move Z to safe position
	eState := eBetriebszustand.Production;
	
	fb_Roboter_Axis_Z.rPosition :=45;
	fb_Roboter_Axis_Z.bExecute :=TRUE;
	bBreak :=TRUE;
	
	IF fb_Roboter_Axis_Z.eState = eBetriebszustand.Done THEN
		fb_Roboter_Axis_Z.bExecute :=FALSE;
		bBreak :=FALSE;
		nstate :=23;
	END_IF
	
	23: //Move xy
	eState := eBetriebszustand.Production;
	
	fb_Roboter_Axis_X.rPosition :=pPositionX;
	fb_Roboter_Axis_X.bExecute :=TRUE;
	fb_Roboter_Axis_Y.rPosition :=pPositionY;
	fb_Roboter_Axis_Y.bExecute :=TRUE;
	
	IF (fb_Roboter_Axis_X.eState = eBetriebszustand.Done) AND (fb_Roboter_Axis_Y.eState = eBetriebszustand.Done) THEN
		fb_Roboter_Axis_X.bExecute :=FALSE;
		fb_Roboter_Axis_Y.bExecute :=FALSE;
		nstate :=24;
	END_IF
	
	24: //Move Z
	eState := eBetriebszustand.Production;
	
	fb_Roboter_Axis_Z.rPosition :=pPositionZ;
	fb_Roboter_Axis_Z.bExecute :=TRUE;
	bBreak :=TRUE;
	
	IF fb_Roboter_Axis_Z.eState = eBetriebszustand.Done THEN
		fb_Roboter_Axis_Z.bExecute :=FALSE;
		bBreak :=FALSE;
		nstate :=25;
	END_IF
	
	25: //Done
	eState := eBetriebszustand.Done;
	
	IF NOT bExecute THEN
		nstate :=2;
	END_IF
	
	
END_CASE

END_FUNCTION_BLOCK

// ---- GlobalTextList.TcGTLO
TEXTLIST GlobalTextList
  747 = '%i'
  734 = 'Betriebszustand'
  0 = 'Betriebszustand %s'
  891 = 'Dispenser1'
  352 = 'Dispenser2'
  700 = 'Dispenser3'
  846 = 'Enable'
  722 = 'Execute'
  977 = 'g'
  204 = 'Rezept'
  143 = 'Status'
  884 = 'Teaching Factory'
  251 = 'Test'
END_TEXTLIST

// ---- VISUs/Visualization.TcVIS
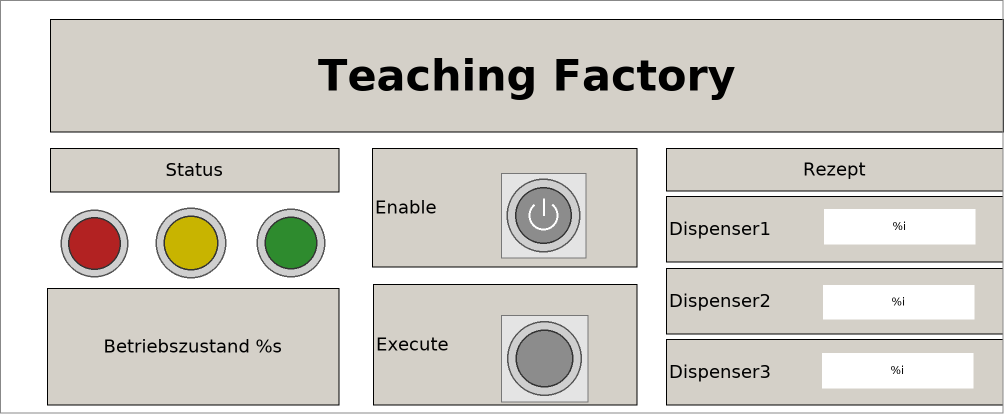
VISUALIZATION Visualization  // 1004x414
    Rectangle (666,196 337x66), "Dispenser1"
    Rectangle (50,19 954x113), "Teaching Factory"
    Lamp1 (55,202 79x83), variable: bAmpelRot, style: Lamp-Lamp1-Red
    Lamp1 (148,202 86x82), variable: bAmpelGelb, style: Lamp-Lamp1-Yellow
    Lamp1 (248,203 86x80), variable: bAmpelGrun, style: Lamp-Lamp1-Green
    Rectangle (50,148 289x44), "Status"
    Textfield (823,208 153x37), "%i", text variable: iBandFullmenge1
        p4168582468: iBandFullmenge1
        OnMouseDown: write the text variable via VisuDialogs.Numpad
    Rectangle (666,268 337x66), "Dispenser2"
    Rectangle (666,339 337x66), "Dispenser3"
    Rectangle (372,148 265x119), "Enable"
    Rectangle (373,284 264x121), "Execute"
    PowerSwitch (501,172 85x87), variable: bEnable, behaviour: TOGGLE, style: Switch-PowerSwitch-Gray
    PushSwitch (501,303 87x111), variable: bExecute, behaviour: TAP, style: Switch-PushSwitch-Gray
    Rectangle (666,148 337x43), "Rezept"
    Rectangle (47,288 292x117), "Betriebszustand %s", text variable: MAIN.fb_Ampelleuchte.eState
    Textfield (822,284 153x36), "%i", text variable: iBandFullmenge2
        p4168582468: iBandFullmenge2
        OnMouseDown: write the text variable via VisuDialogs.Numpad
    Textfield (821,352 153x37), "%i", text variable: iBandFullmenge3
        p4168582468: iBandFullmenge3
        OnMouseDown: write the text variable via VisuDialogs.Numpad
END_VISUALIZATION
